Staubli VAL3: tool.dtx

string pathGun
pointRx pPoint = {wrist=wfree, fatherId=world[0]}
